TYPE ST_CylinderParameters :
STRUCT
	fCylMaxSpeed : LREAL := 0.05; // m/s
END_STRUCT
END_TYPE

(* stored: Version 1.1.0.1, ProductVersion 3.1.4024.12
   DUT ST_CylinderParameters: Id {95d95745-cc46-4445-b9d6-3b9954766e4d} *)
